{attribute 'enable_dynamic_creation'}
FUNCTION_BLOCK FB_ValveMoveCommand IMPLEMENTS I_Command
VAR
	_Valve : I_Valve;
	_Target : E_ValvePosition;
	_Description : STRING;
END_VAR

{attribute 'monitoring' := 'call'}
PROPERTY Description : STRING
GET
Description := _Description;
END_GET
END_PROPERTY

METHOD Execute : E_ProgressStatus
CASE _Target OF
	
	E_ValvePosition.Home:
		_Valve.MoveToHome();
	
	E_ValvePosition.Work:
		_Valve.MoveToWork();
END_CASE

Execute := E_ProgressStatus.Completed;
END_METHOD

//FB_Init is always available implicitly and it is used primarily for initialization.
//The return value is not evaluated. For a specific influence, you can also declare the
//methods explicitly and provide additional code there with the standard initialization
//code. You can evaluate the return value.
METHOD FB_Init: BOOL
VAR_INPUT
    bInitRetains: BOOL; // TRUE: the retain variables are initialized (reset warm / reset cold)
    bInCopyCode: BOOL;  // TRUE: the instance will be copied to the copy code afterward (online change)   
	
	valve : I_Valve;
	target : E_ValvePosition;
	description : STRING;
END_VAR
_Valve := valve;
_Target := target;
_Description := description;
END_METHOD

METHOD Reset
VAR_INPUT
END_VAR
// nothing to reset here
END_METHOD

END_FUNCTION_BLOCK

(* stored: Version 1.1.0.1
   POU FB_ValveMoveCommand: Id {047c86e1-dcc4-4b85-9610-35c466eed17c}, SpecialFunc None
   Property Description: Id {cbf14950-4b79-4d96-ab7a-2f398e37eb22}
   Get Get: Id {e59c0537-ef0f-4533-9f3e-d3b6d2ebbafb}
   Method Execute: Id {4d5ed5e8-4bdd-4c01-8be0-e7a4f0af3875}
   Method FB_Init: Id {77fb1ac3-10bd-4baa-9eec-c07e022e78d0}
   Method Reset: Id {19a3253b-3ef6-43be-bbbe-973700a5a543} *)
